RoboDK station: DrawingProject.rdk

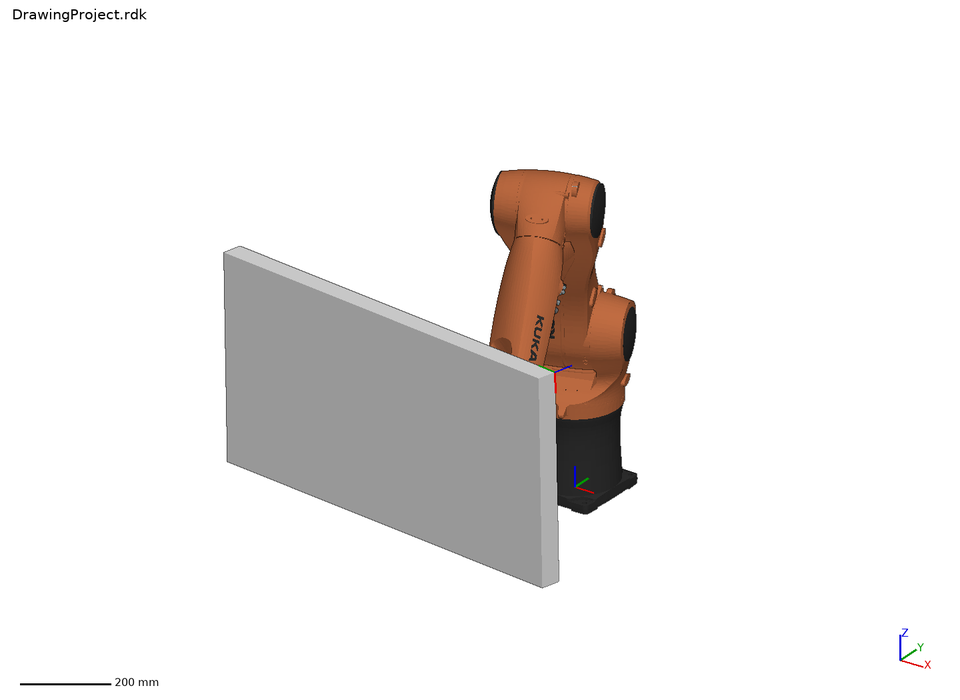
[picture v0: the station drawn from its stored meshes, robots at their saved joint values, targets as dots, program paths as lines]
Station DrawingProject (saved by RoboDK 5.2.1). Poses are relative to the parent item; angles as X-Y-Z fixed-axis rotations.
  - frame KUKA KR 6 R900 sixx Base at (0, 0, 0) mm
    - robot KUKA KR 6 R900 sixx: 6 axes, payload 6 kg, reach 901 mm, repeatability 0.03 mm, weight 52 kg
        modified DH rows (alpha deg, a mm, theta deg, d mm): 0, 0, 0, 400; -90, 25, 0, 0; 0, 455, -90, 0; -90, 35, 0, 420; 90, 0, 0, 0; -90, 0, 180, 80
        joint limits [-170, -190, -120, -185, -120, -350] to [170, 45, 156, 185, 120, 350]; home [0, -90, 90, 0, 0, 0]; saved at [68.709, -61.721, 105.379, 137.935, 53.424, 26.503]
      - tool Assemb_Base2_Marker-Part, TCP at (0, 0, 128) mm, size 40 x 40 x 147.5 mm, geometry from Assemb_Base2_Marker-Part.stl
    - object pixel at (0, 0, 0) mm, size 10 x 10 x 1 mm
  - frame Frame draw at (482.33, -764.55, 720.57) mm, rotated rx -114.61 ry 87.25 rz -35.85 deg
    - object Blackboard 250mm at (0, 0, 0) mm, size 250 x 250 x 50 mm
    - object Board & image at (0, 0, 0) mm, size 500 x 1000 x 50 mm
